(* Logix 5000 project; controller AMANA_DC_PLANT_01 vendor 1 type 14 code 164 rev 31.12; software revision 31.02; part 6 of 9 *)
(* tags used below, declared in another part *)
   badModel : STRING_40;
   Break_1stStation : BOOL;
   firstCharacter : STRING_40;
   Local_Timer : TIMER[10];
   OneShot : DINT;
   ONS_20 : DINT;
   previousSerialNumber : STRING;
   readIndex : DINT;
   tempIndex : DINT;
   writeIndex : DINT;
   DC1_OPCFault : BOOL;
   DC1_to_LN00_Messages : DINT[20];
   DC1_to_LN00_Time_sync_Out : MESSAGE;
   LN00_COUNTS_FROM_IGN_DB_msg : MESSAGE;
   LN00_MainLine_MSG_Out : MESSAGE;
   LN00_Schedule : UDT_Current_Status;
   LN00_SNModel_Array : UDT_SN_Model[50];
   LN00_SNModel_CurrentRead : UDT_SN_Model;
   LN00_SNModel_STR : STRING[10];
   LN00_to_DC1_Main_Messages_6 : DINT[120];
   LN00DFM04 : DINT;
   LN00DFM05 : DINT;
   LN00DFM06 : DINT;
   LN00DFM07 : DINT;
   LN00DFM08 : DINT;
   LN00DFM09 : DINT;
   LN00DFM10 : DINT;
   LN00DFM11 : DINT;
   LN00DFM12 : DINT;
   LN00DFM13 : DINT;
   LN00DFM14 : DINT;
   LN00DFM15 : DINT;
   LN00DFM16 : DINT;
   LN00DFM17 : DINT;
   LN00DFM18 : DINT;
   LN00DFM19 : DINT;
   LN00DFM20 : DINT;
   LN00DFM21 : DINT;
   LN00DFM22 : DINT;
   LN00DFM23 : DINT;
   LN00DFM24 : DINT;
   LN00DFM25 : DINT;
   LN00DFM26 : DINT;
   LN00DFM27 : DINT;
   LN00DFM28 : DINT;
   LN00DFM29 : DINT;
   LN00DFM30 : DINT;
   LN00DFM31 : DINT;
   LN00DFM32 : DINT;
   LN00DFM33 : DINT;
   LN00DFM34 : DINT;
   LN00DFM35 : DINT;
   msg192_reset_timer : TIMER;
   null : STRING;
   OH_Barcode_Model_CLEARPACK : STRING;
   OH_Barcode_Model_DOCKSORTING : STRING;
   OH_Barcode_Model_LN4 : STRING;
   OH_Barcode_Model_LN467MERGE : STRING;
   OH_Barcode_Model_LN6 : STRING;
   OH_Barcode_Model_LN67MERGE : STRING;
   OH_Barcode_Model_LN7 : STRING;
   OH_Barcode_Model_LONGTERMEAST : STRING;
   OH_Barcode_Model_LONGTERMWEST : STRING;
   OH_Barcode_Model_WAREHOUSENORTH : STRING;
   OH_Barcode_Model_WAREHOUSESOUTH : STRING;
   OH_Barcode_Serial_CLEARPACK : STRING;
   OH_Barcode_Serial_DOCKSORTING : STRING;
   OH_Barcode_Serial_LN4 : STRING;
   OH_Barcode_Serial_LN467MERGE : STRING;
   OH_Barcode_Serial_LN6 : STRING;
   OH_Barcode_Serial_LN67MERGE : STRING;
   OH_Barcode_Serial_LN7 : STRING;
   OH_Barcode_Serial_LONGTERMEAST : STRING;
   OH_Barcode_Serial_LONGTERMWEST : STRING;
   OH_Barcode_Serial_WAREHOUSENORTH : STRING;
   OH_Barcode_Serial_WAREHOUSESOUTH : STRING;
   Shift_reset_timer : TIMER;
(* LN00, continued *)

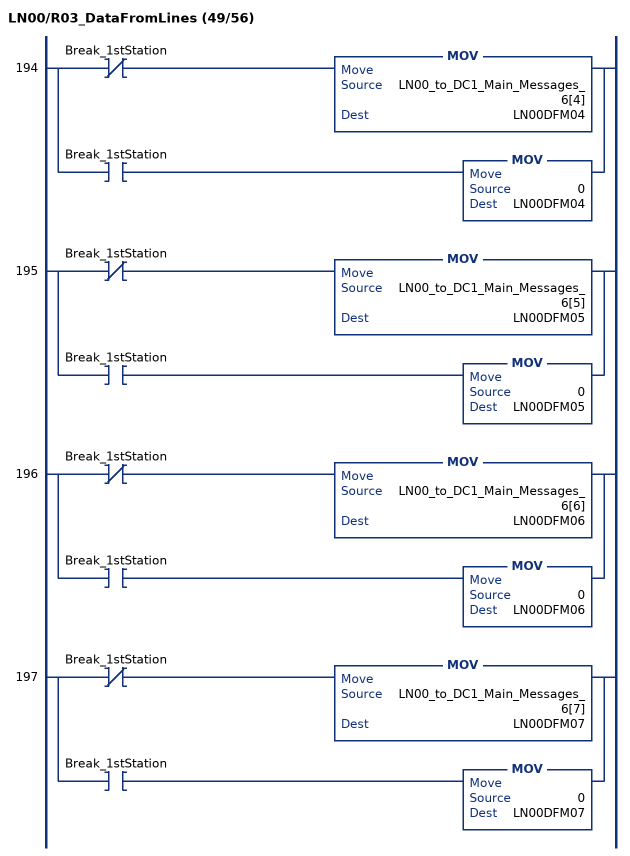
   [picture p95: LN00/R03_DataFromLines rungs 194-197]
   194: [XIO(Break_1stStation) MOV(LN00_to_DC1_Main_Messages_6[4],LN00DFM04) ,XIC(Break_1stStation) MOV(0,LN00DFM04) ];
   195: [XIO(Break_1stStation) MOV(LN00_to_DC1_Main_Messages_6[5],LN00DFM05) ,XIC(Break_1stStation) MOV(0,LN00DFM05) ];
   196: [XIO(Break_1stStation) MOV(LN00_to_DC1_Main_Messages_6[6],LN00DFM06) ,XIC(Break_1stStation) MOV(0,LN00DFM06) ];
   197: [XIO(Break_1stStation) MOV(LN00_to_DC1_Main_Messages_6[7],LN00DFM07) ,XIC(Break_1stStation) MOV(0,LN00DFM07) ];
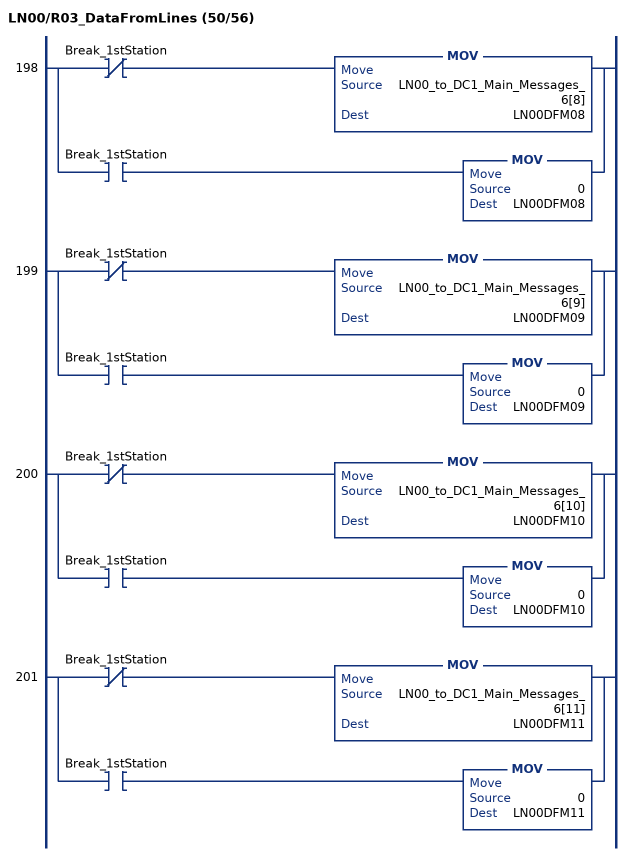
   198: [XIO(Break_1stStation) MOV(LN00_to_DC1_Main_Messages_6[8],LN00DFM08) ,XIC(Break_1stStation) MOV(0,LN00DFM08) ];
   199: [XIO(Break_1stStation) MOV(LN00_to_DC1_Main_Messages_6[9],LN00DFM09) ,XIC(Break_1stStation) MOV(0,LN00DFM09) ];
   200: [XIO(Break_1stStation) MOV(LN00_to_DC1_Main_Messages_6[10],LN00DFM10) ,XIC(Break_1stStation) MOV(0,LN00DFM10) ];
   201: [XIO(Break_1stStation) MOV(LN00_to_DC1_Main_Messages_6[11],LN00DFM11) ,XIC(Break_1stStation) MOV(0,LN00DFM11) ];
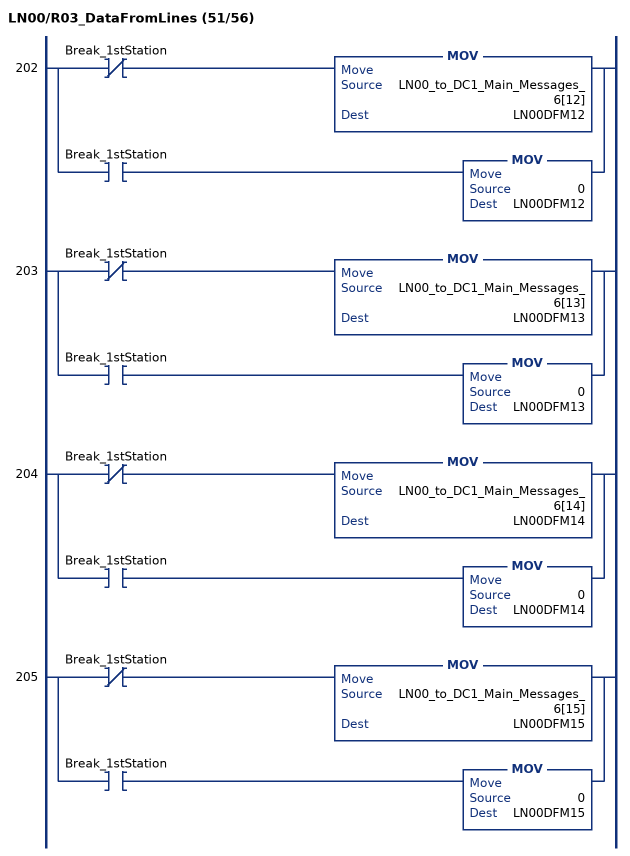
   202: [XIO(Break_1stStation) MOV(LN00_to_DC1_Main_Messages_6[12],LN00DFM12) ,XIC(Break_1stStation) MOV(0,LN00DFM12) ];
   203: [XIO(Break_1stStation) MOV(LN00_to_DC1_Main_Messages_6[13],LN00DFM13) ,XIC(Break_1stStation) MOV(0,LN00DFM13) ];
   204: [XIO(Break_1stStation) MOV(LN00_to_DC1_Main_Messages_6[14],LN00DFM14) ,XIC(Break_1stStation) MOV(0,LN00DFM14) ];
   205: [XIO(Break_1stStation) MOV(LN00_to_DC1_Main_Messages_6[15],LN00DFM15) ,XIC(Break_1stStation) MOV(0,LN00DFM15) ];
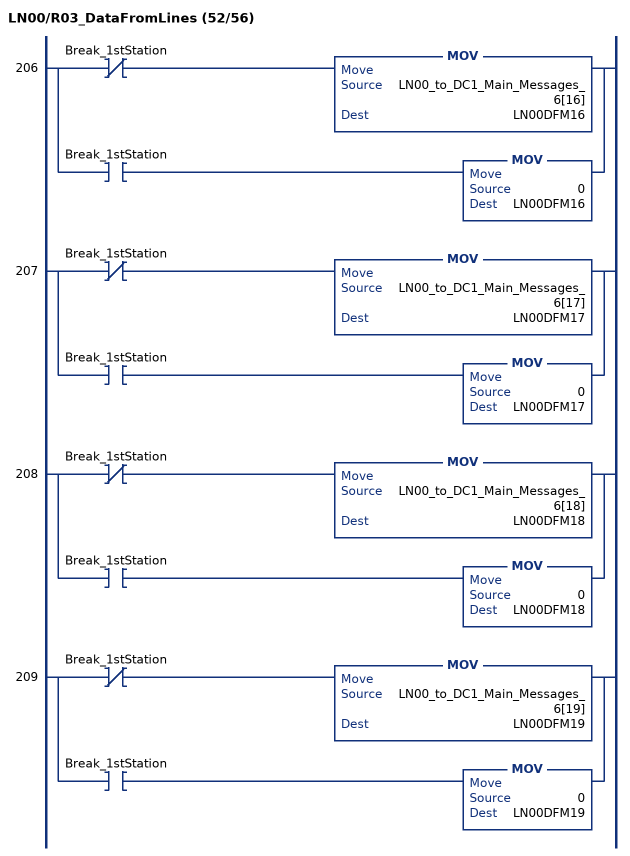
   206: [XIO(Break_1stStation) MOV(LN00_to_DC1_Main_Messages_6[16],LN00DFM16) ,XIC(Break_1stStation) MOV(0,LN00DFM16) ];
   207: [XIO(Break_1stStation) MOV(LN00_to_DC1_Main_Messages_6[17],LN00DFM17) ,XIC(Break_1stStation) MOV(0,LN00DFM17) ];
   208: [XIO(Break_1stStation) MOV(LN00_to_DC1_Main_Messages_6[18],LN00DFM18) ,XIC(Break_1stStation) MOV(0,LN00DFM18) ];
   209: [XIO(Break_1stStation) MOV(LN00_to_DC1_Main_Messages_6[19],LN00DFM19) ,XIC(Break_1stStation) MOV(0,LN00DFM19) ];
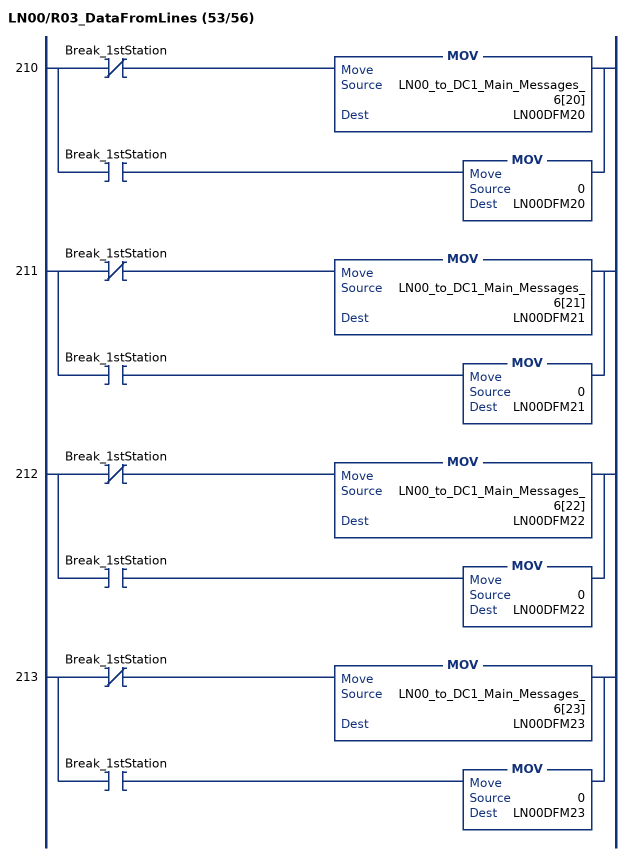
   210: [XIO(Break_1stStation) MOV(LN00_to_DC1_Main_Messages_6[20],LN00DFM20) ,XIC(Break_1stStation) MOV(0,LN00DFM20) ];
   211: [XIO(Break_1stStation) MOV(LN00_to_DC1_Main_Messages_6[21],LN00DFM21) ,XIC(Break_1stStation) MOV(0,LN00DFM21) ];
   212: [XIO(Break_1stStation) MOV(LN00_to_DC1_Main_Messages_6[22],LN00DFM22) ,XIC(Break_1stStation) MOV(0,LN00DFM22) ];
   213: [XIO(Break_1stStation) MOV(LN00_to_DC1_Main_Messages_6[23],LN00DFM23) ,XIC(Break_1stStation) MOV(0,LN00DFM23) ];
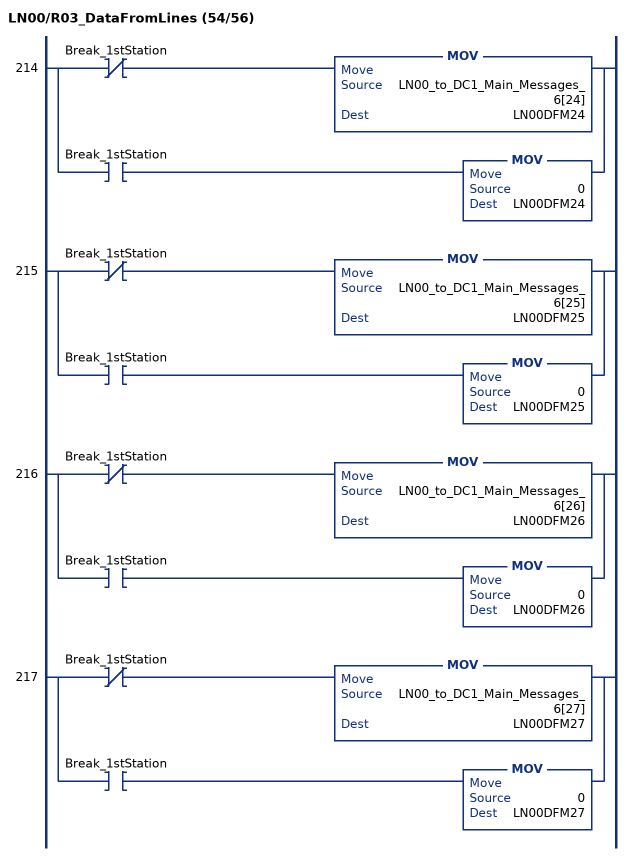
   214: [XIO(Break_1stStation) MOV(LN00_to_DC1_Main_Messages_6[24],LN00DFM24) ,XIC(Break_1stStation) MOV(0,LN00DFM24) ];
   215: [XIO(Break_1stStation) MOV(LN00_to_DC1_Main_Messages_6[25],LN00DFM25) ,XIC(Break_1stStation) MOV(0,LN00DFM25) ];
   216: [XIO(Break_1stStation) MOV(LN00_to_DC1_Main_Messages_6[26],LN00DFM26) ,XIC(Break_1stStation) MOV(0,LN00DFM26) ];
   217: [XIO(Break_1stStation) MOV(LN00_to_DC1_Main_Messages_6[27],LN00DFM27) ,XIC(Break_1stStation) MOV(0,LN00DFM27) ];
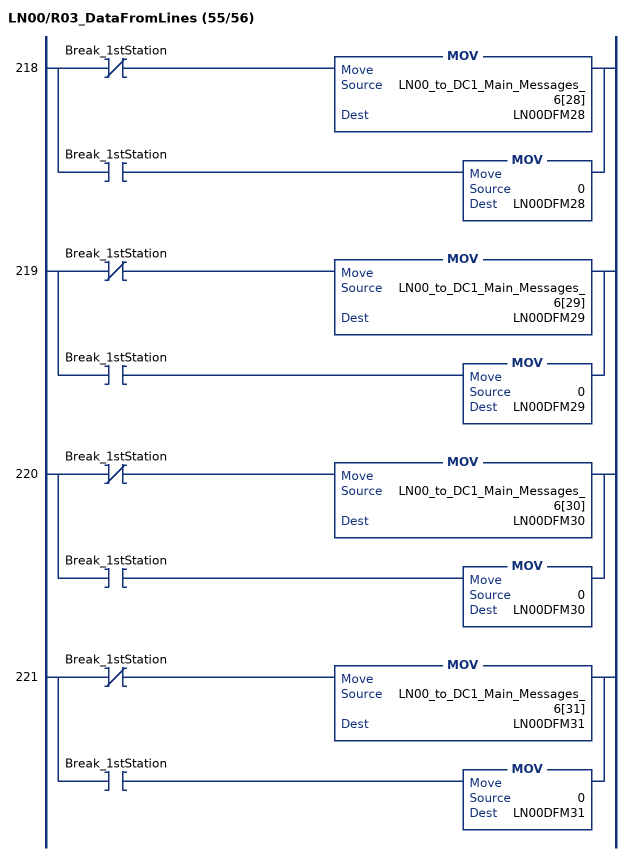
   218: [XIO(Break_1stStation) MOV(LN00_to_DC1_Main_Messages_6[28],LN00DFM28) ,XIC(Break_1stStation) MOV(0,LN00DFM28) ];
   219: [XIO(Break_1stStation) MOV(LN00_to_DC1_Main_Messages_6[29],LN00DFM29) ,XIC(Break_1stStation) MOV(0,LN00DFM29) ];
   220: [XIO(Break_1stStation) MOV(LN00_to_DC1_Main_Messages_6[30],LN00DFM30) ,XIC(Break_1stStation) MOV(0,LN00DFM30) ];
   221: [XIO(Break_1stStation) MOV(LN00_to_DC1_Main_Messages_6[31],LN00DFM31) ,XIC(Break_1stStation) MOV(0,LN00DFM31) ];
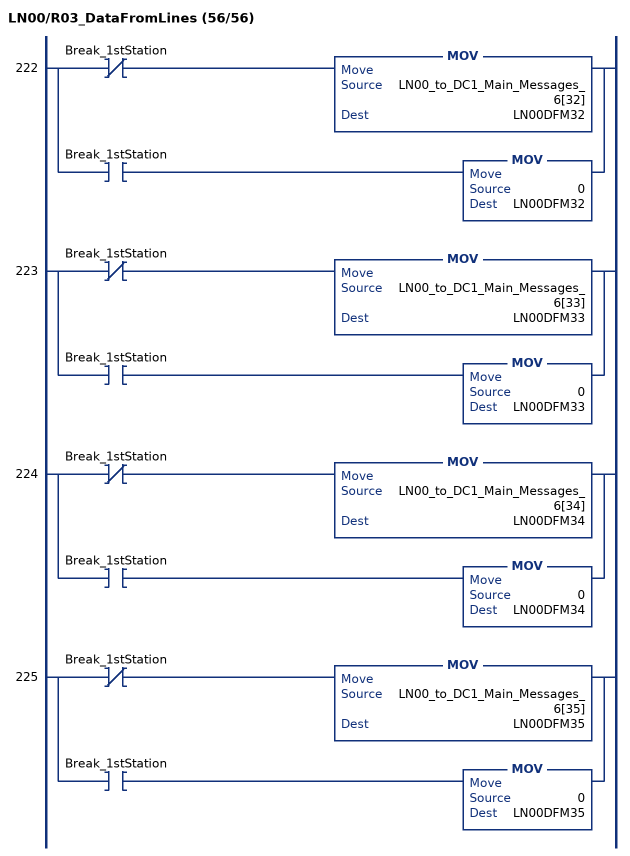
   222: [XIO(Break_1stStation) MOV(LN00_to_DC1_Main_Messages_6[32],LN00DFM32) ,XIC(Break_1stStation) MOV(0,LN00DFM32) ];
   223: [XIO(Break_1stStation) MOV(LN00_to_DC1_Main_Messages_6[33],LN00DFM33) ,XIC(Break_1stStation) MOV(0,LN00DFM33) ];
   224: [XIO(Break_1stStation) MOV(LN00_to_DC1_Main_Messages_6[34],LN00DFM34) ,XIC(Break_1stStation) MOV(0,LN00DFM34) ];
   225: [XIO(Break_1stStation) MOV(LN00_to_DC1_Main_Messages_6[35],LN00DFM35) ,XIC(Break_1stStation) MOV(0,LN00DFM35) ];
END_ROUTINE

ROUTINE R04_DataToLines   (* ladder *)
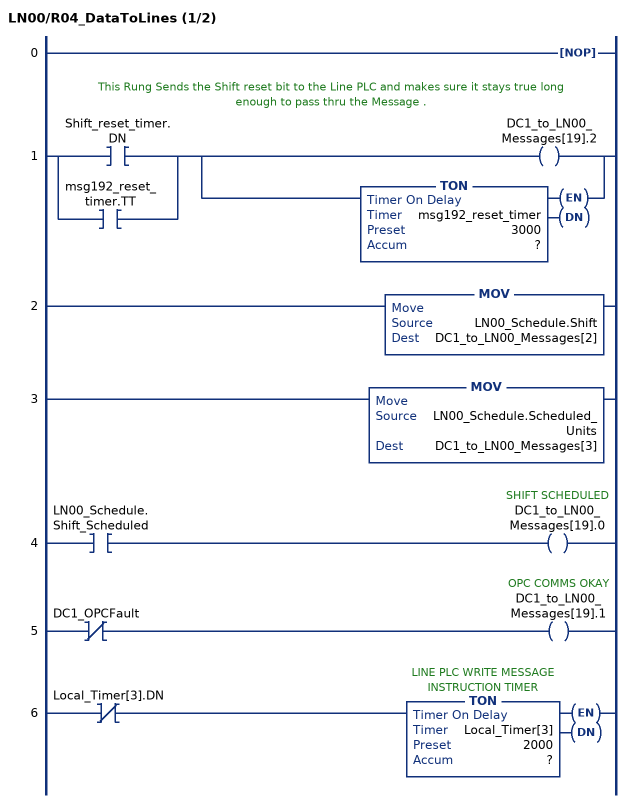
   0: NOP();
   // This Rung Sends the Shift reset bit to the Line PLC and makes sure it stays true long enough to pass thru the Message .
   1: [XIC(Shift_reset_timer.DN) ,XIC(msg192_reset_timer.TT) ][OTE(DC1_to_LN00_Messages[19].2) ,TON(msg192_reset_timer,?,?) ];
   2: MOV(LN00_Schedule.Shift,DC1_to_LN00_Messages[2]);
   3: MOV(LN00_Schedule.Scheduled_Units,DC1_to_LN00_Messages[3]);
   4: XIC(LN00_Schedule.Shift_Scheduled)OTE(DC1_to_LN00_Messages[19].0);
   5: XIO(DC1_OPCFault)OTE(DC1_to_LN00_Messages[19].1);
   6: XIO(Local_Timer[3].DN)TON(Local_Timer[3],?,?);
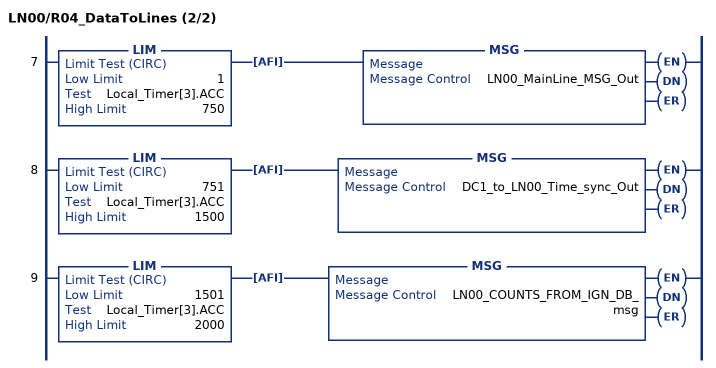
   7: LIM(1,Local_Timer[3].ACC,750)AFI()MSG(LN00_MainLine_MSG_Out);
   8: LIM(751,Local_Timer[3].ACC,1500)AFI()MSG(DC1_to_LN00_Time_sync_Out);
   9: LIM(1501,Local_Timer[3].ACC,2000)AFI()MSG(LN00_COUNTS_FROM_IGN_DB_msg);
END_ROUTINE

ROUTINE R05_SNModel_Manager   (* ladder *)
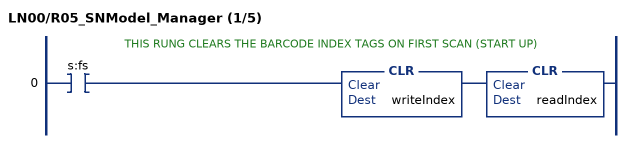
   // THIS RUNG CLEARS THE BARCODE INDEX TAGS ON FIRST SCAN (START UP)
   0: XIC(s:fs)CLR(writeIndex)CLR(readIndex);
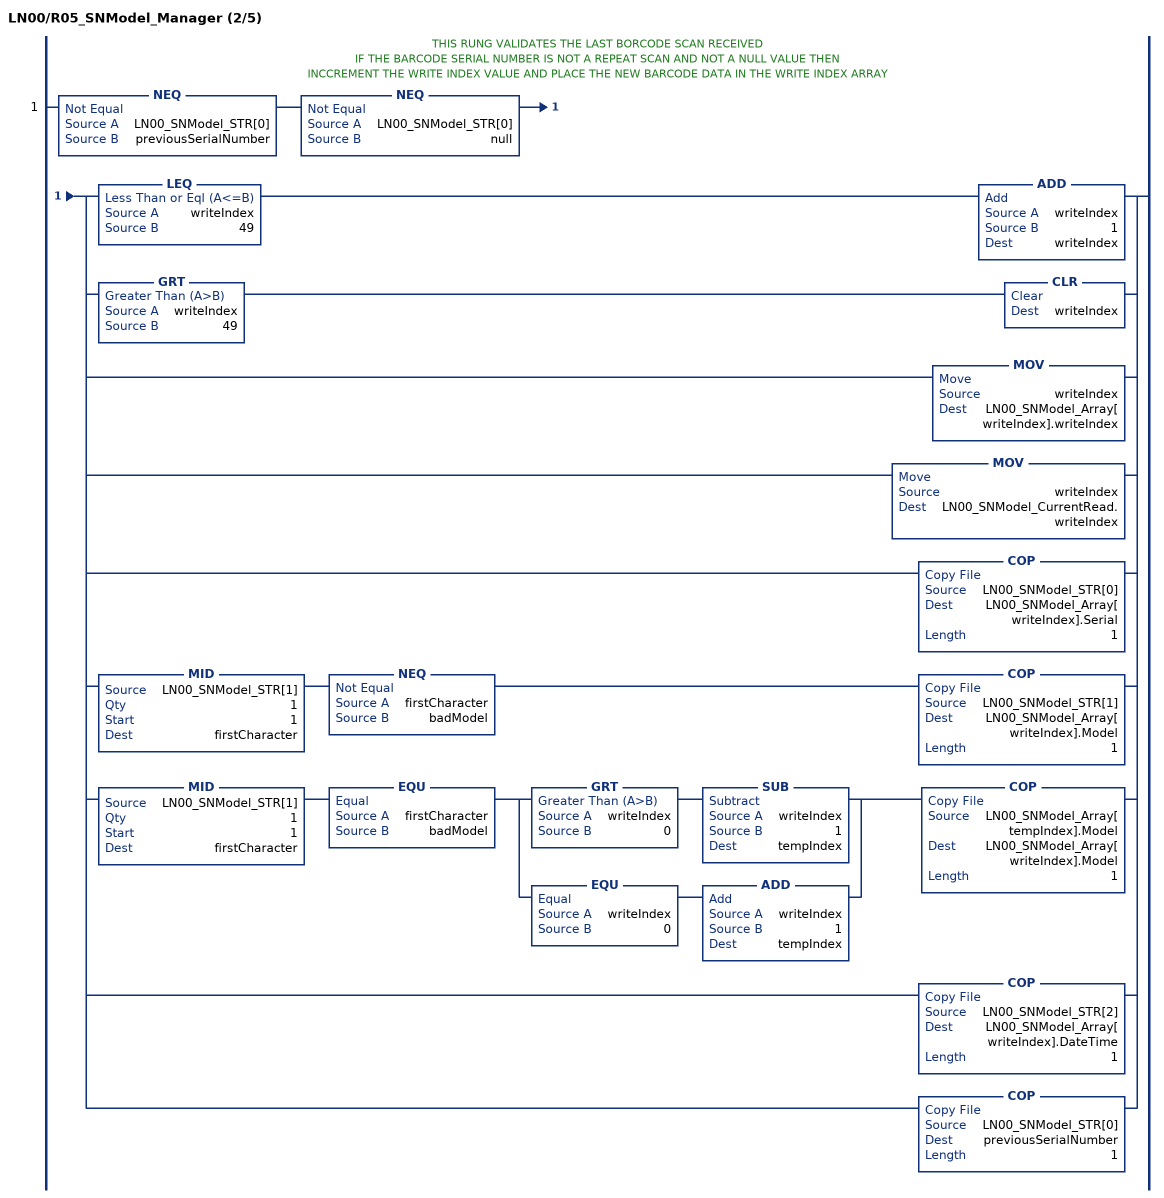
   // THIS RUNG VALIDATES THE LAST BORCODE SCAN RECEIVED
   // IF THE BARCODE SERIAL NUMBER IS NOT A REPEAT SCAN AND NOT A NULL VALUE THEN
   // INCCREMENT THE WRITE INDEX VALUE AND PLACE THE NEW BARCODE DATA IN THE WRITE INDEX ARRAY
   1: NEQ(LN00_SNModel_STR[0],previousSerialNumber)NEQ(LN00_SNModel_STR[0],null)[[LEQ(writeIndex,49) ADD(writeIndex,1,writeIndex) ,GRT(writeIndex,49) CLR(writeIndex) ,MOV(writeIndex,LN00_SNModel_Array[writeIndex].writeIndex) ,MOV(writeIndex,LN00_SNModel_CurrentRead.writeIndex) ,COP(LN00_SNModel_STR[0],LN00_SNModel_Array[writeIndex].Serial,1) ,MID(LN00_SNModel_STR[1],1,1,firstCharacter) NEQ(firstCharacter,badModel) COP(LN00_SNModel_STR[1],LN00_SNModel_Array[writeIndex].Model,1) ,MID(LN00_SNModel_STR[1],1,1,firstCharacter) EQU(firstCharacter,badModel) [GRT(writeIndex,0) SUB(writeIndex,1,tempIndex) ,EQU(writeIndex,0) ADD(writeIndex,1,tempIndex) ] COP(LN00_SNModel_Array[tempIndex].Model,LN00_SNModel_Array[writeIndex].Model,1) ,COP(LN00_SNModel_STR[2],LN00_SNModel_Array[writeIndex].DateTime,1) ] ,COP(LN00_SNModel_STR[0],previousSerialNumber,1) ];
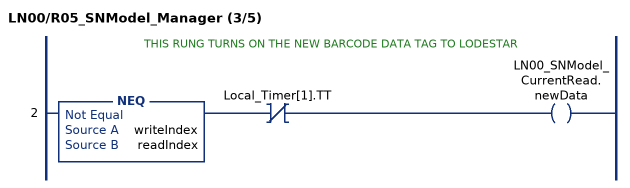
   // THIS RUNG TURNS ON THE NEW BARCODE DATA TAG TO LODESTAR
   2: NEQ(writeIndex,readIndex)XIO(Local_Timer[1].TT)OTE(LN00_SNModel_CurrentRead.newData);
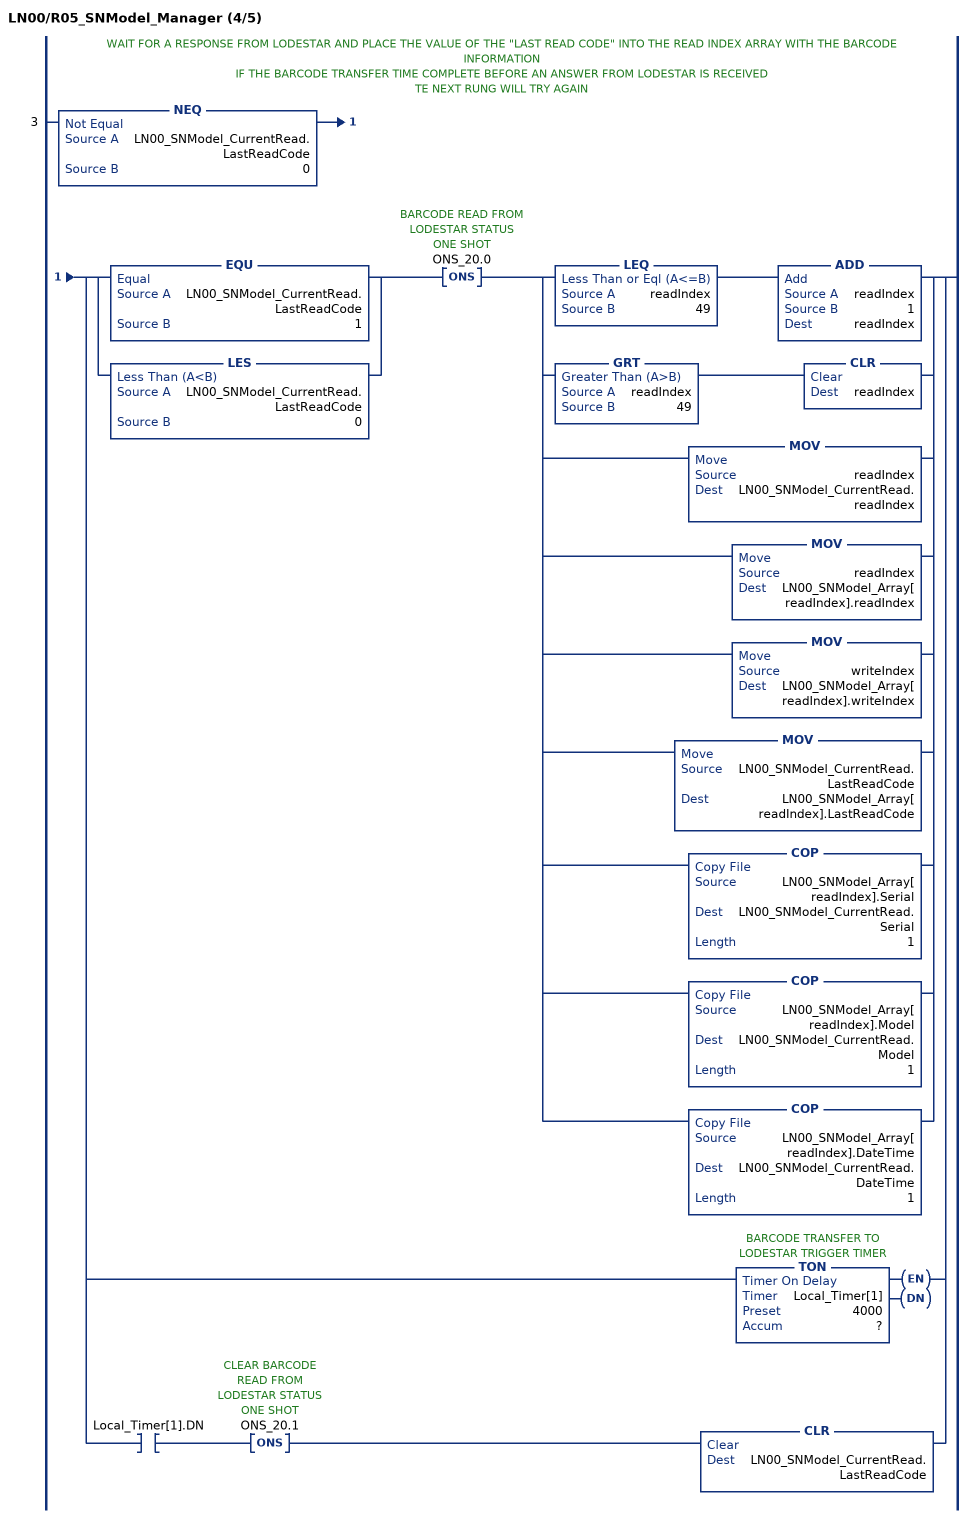
   // WAIT FOR A RESPONSE FROM LODESTAR AND PLACE THE VALUE OF THE "LAST READ CODE" INTO THE READ INDEX ARRAY WITH THE BARCODE INFORMATION
   // IF THE BARCODE TRANSFER TIME COMPLETE BEFORE AN ANSWER FROM LODESTAR IS RECEIVED
   // TE NEXT RUNG WILL TRY AGAIN
   3: NEQ(LN00_SNModel_CurrentRead.LastReadCode,0)[[EQU(LN00_SNModel_CurrentRead.LastReadCode,1) ,LES(LN00_SNModel_CurrentRead.LastReadCode,0) ] ONS(ONS_20.0) [LEQ(readIndex,49) ADD(readIndex,1,readIndex) ,GRT(readIndex,49) CLR(readIndex) ,MOV(readIndex,LN00_SNModel_CurrentRead.readIndex) ,MOV(readIndex,LN00_SNModel_Array[readIndex].readIndex) ,MOV(writeIndex,LN00_SNModel_Array[readIndex].writeIndex) ,MOV(LN00_SNModel_CurrentRead.LastReadCode,LN00_SNModel_Array[readIndex].LastReadCode) ,COP(LN00_SNModel_Array[readIndex].Serial,LN00_SNModel_CurrentRead.Serial,1) ,COP(LN00_SNModel_Array[readIndex].Model,LN00_SNModel_CurrentRead.Model,1) ,COP(LN00_SNModel_Array[readIndex].DateTime,LN00_SNModel_CurrentRead.DateTime,1) ] ,[TON(Local_Timer[1],?,?) ,XIC(Local_Timer[1].DN) ONS(ONS_20.1) CLR(LN00_SNModel_CurrentRead.LastReadCode) ] ];
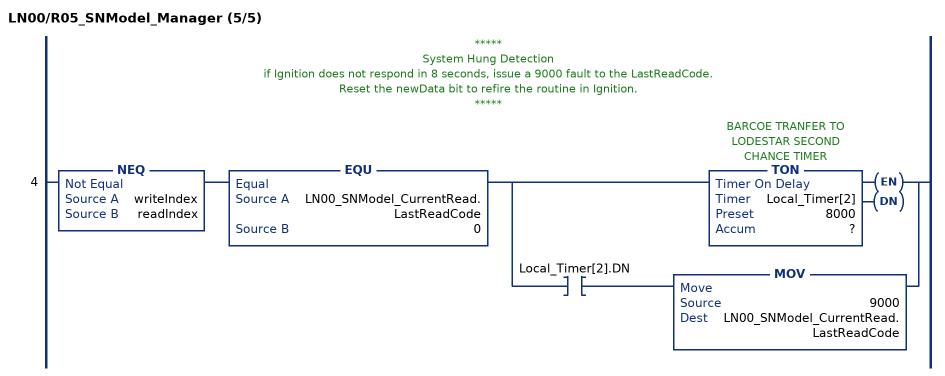
   // *****
   // System Hung Detection
   // if Ignition does not respond in 8 seconds, issue a 9000 fault to the LastReadCode.
   // Reset the newData bit to refire the routine in Ignition.
   // *****
   4: NEQ(writeIndex,readIndex)EQU(LN00_SNModel_CurrentRead.LastReadCode,0)[TON(Local_Timer[2],?,?) ,XIC(Local_Timer[2].DN) MOV(9000,LN00_SNModel_CurrentRead.LastReadCode) ];
END_ROUTINE
END_PROGRAM

PROGRAM OH_BARCODE_SCAN   (* main routine R00_Main *)
VAR
   Barcode_Longest : DINT := 24;
   Barcode_Shortest : DINT := 20;
   Comma : STRING := ',';
   Counters : COUNTER[16] := ([1].PRE := 3, [2].DN := 1, [3].DN := 1, [4].DN := 1, [5].DN := 1, [6].DN := 1);
        [1]   // ClearPack MSG 1 Error Counter
   MSG_Enable : DINT := 34;
   MSG_ONS : DINT := 4;
   MSG_Steps : DINT := 2;
   NULL_String : STRING;
   PRE_SET_COMMA_POSITION_1 : DINT := 12;
   SCANNER_ClearPack_DATA : Keyence_2_Barcode := (Trigger_Timer.PRE := 500, Barcode_ReadIsSuccess := 1, Barcode_Raw := 'WRB322DMBM 03,KC1814086', Barcode_Comma_Position := 14, Barcode_1_Length := 13, Barcode_2_Length := 9, Barcode_2_Start := 15, Barcode_1_String := 'WRB322DMBM 03', Barcode_2_String := 'KC1814086', Barcode_SRReaderReady := 1);
   SCANNER_DOCKSORTING_DATA : Keyence_2_Barcode := (Trigger_Timer.PRE := 200, Trigger_Timer.EN := 1, Trigger_Timer.DN := 1, Barcode_SRTrigger := 1, Barcode_Comma_Position := 10, Barcode_1_Length := 9, Barcode_2_Length := 13, Barcode_2_Start := 11, PlaceHolder_ConveyorRunning := 1, OneShot := 1);
   SCANNER_LN467MERGE_DATA : Keyence_2_Barcode := (Trigger_Timer.PRE := 200, Trigger_Timer.ACC := 200, OneShot := 1);
   SCANNER_LN4_DATA : Keyence_2_Barcode := (Trigger_Timer.PRE := 200, Trigger_Timer.ACC := 200, OneShot := 1);
   SCANNER_LN67MERGE_DATA : Keyence_2_Barcode := (Trigger_Timer.PRE := 200, Trigger_Timer.ACC := 200, OneShot := 1);
   SCANNER_LN6_DATA : Keyence_2_Barcode := (Trigger_Timer.PRE := 200, Trigger_Timer.ACC := 200, OneShot := 1);
   SCANNER_LN7_DATA : Keyence_2_Barcode := (Trigger_Timer.PRE := 200, Trigger_Timer.ACC := 200, OneShot := 1);
   SCANNER_LONGTERMEAST_DATA : Keyence_2_Barcode := (Trigger_Timer.PRE := 200, Trigger_Timer.ACC := 200, OneShot := 1);
   SCANNER_LONGTERMWEST_DATA : Keyence_2_Barcode := (Trigger_Timer.PRE := 200, Trigger_Timer.ACC := 200, OneShot := 1);
   SCANNER_WAREHOUSENORTH_DATA : Keyence_2_Barcode := (Trigger_Timer.PRE := 200, Trigger_Timer.ACC := 200, OneShot := 1);
   SCANNER_WAREHOUSESOUTH_DATA : Keyence_2_Barcode := (Trigger_Timer.PRE := 200, Trigger_Timer.ACC := 200, OneShot := 1);
   Test_Bits : DINT := 2051;
   Timer_MSG_Interval : TIMER := (PRE := 500);
END_VAR

ROUTINE R00_Main   (* ladder *)
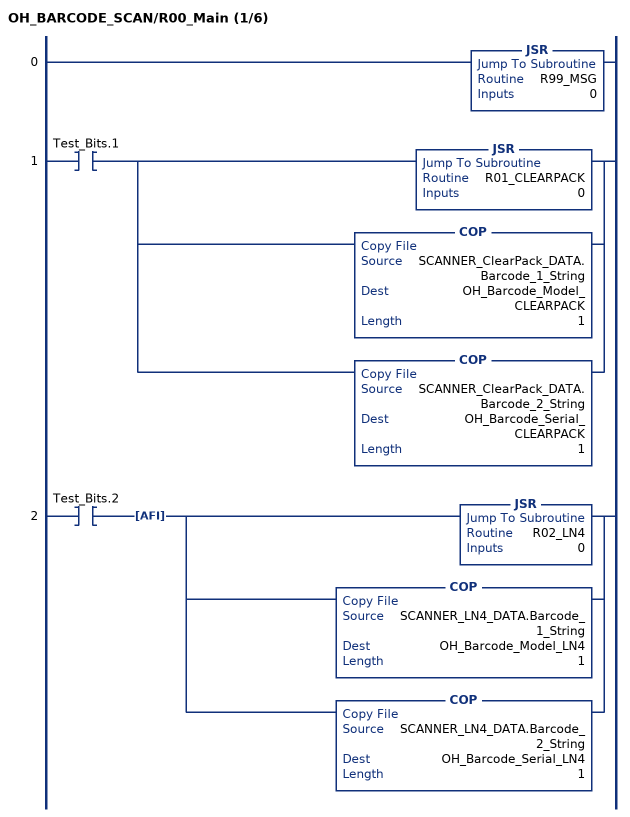
   0: JSR(R99_MSG,0);
   1: XIC(Test_Bits.1)[JSR(R01_CLEARPACK,0) ,COP(SCANNER_ClearPack_DATA.Barcode_1_String,OH_Barcode_Model_CLEARPACK,1) ,COP(SCANNER_ClearPack_DATA.Barcode_2_String,OH_Barcode_Serial_CLEARPACK,1) ];
   2: XIC(Test_Bits.2)AFI()[JSR(R02_LN4,0) ,COP(SCANNER_LN4_DATA.Barcode_1_String,OH_Barcode_Model_LN4,1) ,COP(SCANNER_LN4_DATA.Barcode_2_String,OH_Barcode_Serial_LN4,1) ];
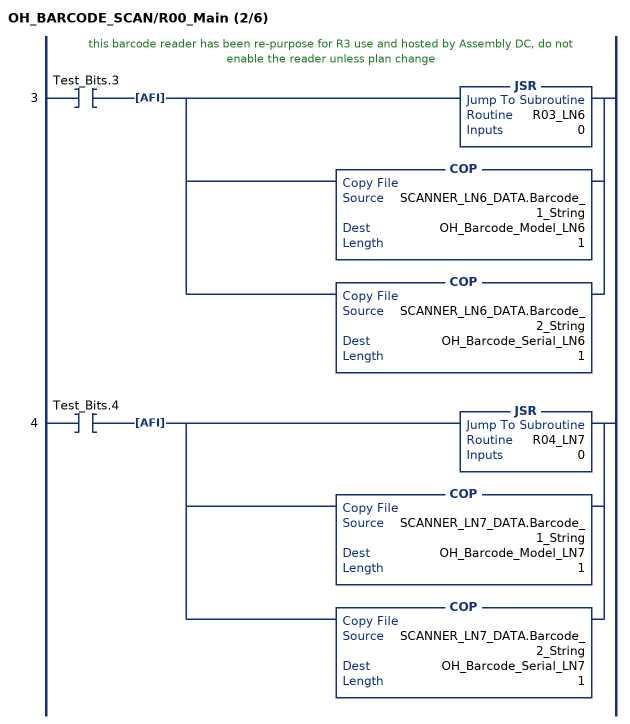
   // this barcode reader has been re-purpose for R3 use and hosted by Assembly DC, do not enable the reader unless plan change
   3: XIC(Test_Bits.3)AFI()[JSR(R03_LN6,0) ,COP(SCANNER_LN6_DATA.Barcode_1_String,OH_Barcode_Model_LN6,1) ,COP(SCANNER_LN6_DATA.Barcode_2_String,OH_Barcode_Serial_LN6,1) ];
   4: XIC(Test_Bits.4)AFI()[JSR(R04_LN7,0) ,COP(SCANNER_LN7_DATA.Barcode_1_String,OH_Barcode_Model_LN7,1) ,COP(SCANNER_LN7_DATA.Barcode_2_String,OH_Barcode_Serial_LN7,1) ];
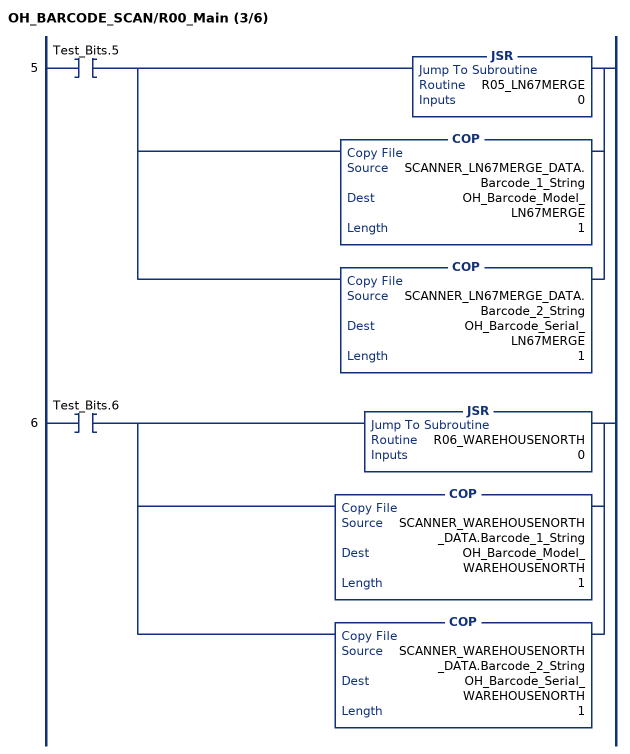
   5: XIC(Test_Bits.5)[JSR(R05_LN67MERGE,0) ,COP(SCANNER_LN67MERGE_DATA.Barcode_1_String,OH_Barcode_Model_LN67MERGE,1) ,COP(SCANNER_LN67MERGE_DATA.Barcode_2_String,OH_Barcode_Serial_LN67MERGE,1) ];
   6: XIC(Test_Bits.6)[JSR(R06_WAREHOUSENORTH,0) ,COP(SCANNER_WAREHOUSENORTH_DATA.Barcode_1_String,OH_Barcode_Model_WAREHOUSENORTH,1) ,COP(SCANNER_WAREHOUSENORTH_DATA.Barcode_2_String,OH_Barcode_Serial_WAREHOUSENORTH,1) ];
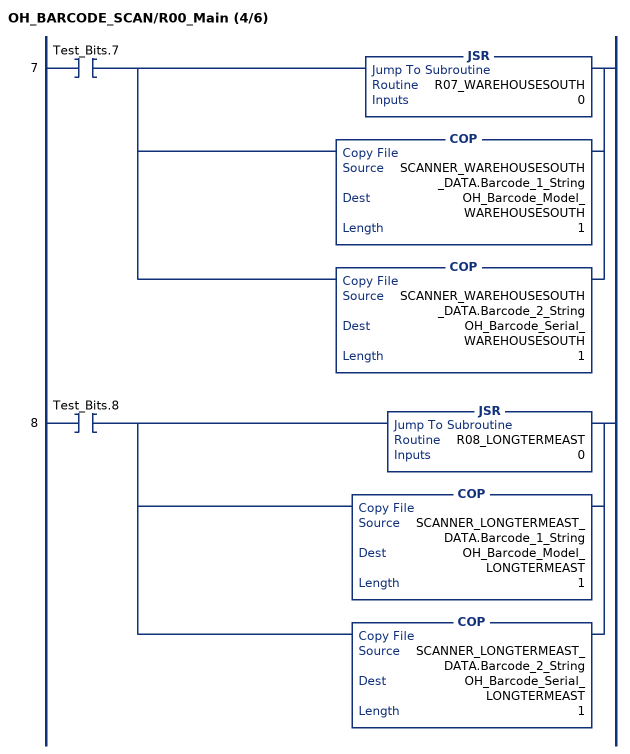
   7: XIC(Test_Bits.7)[JSR(R07_WAREHOUSESOUTH,0) ,COP(SCANNER_WAREHOUSESOUTH_DATA.Barcode_1_String,OH_Barcode_Model_WAREHOUSESOUTH,1) ,COP(SCANNER_WAREHOUSESOUTH_DATA.Barcode_2_String,OH_Barcode_Serial_WAREHOUSESOUTH,1) ];
   8: XIC(Test_Bits.8)[JSR(R08_LONGTERMEAST,0) ,COP(SCANNER_LONGTERMEAST_DATA.Barcode_1_String,OH_Barcode_Model_LONGTERMEAST,1) ,COP(SCANNER_LONGTERMEAST_DATA.Barcode_2_String,OH_Barcode_Serial_LONGTERMEAST,1) ];
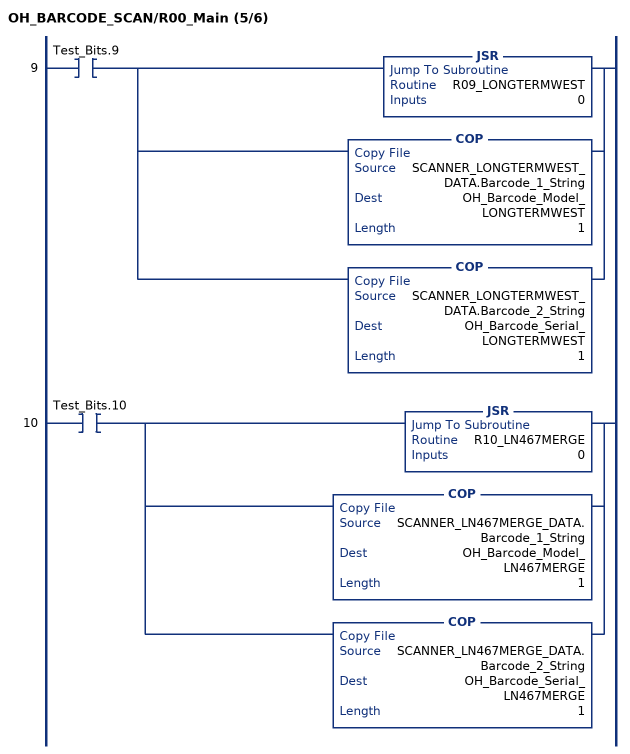
   9: XIC(Test_Bits.9)[JSR(R09_LONGTERMWEST,0) ,COP(SCANNER_LONGTERMWEST_DATA.Barcode_1_String,OH_Barcode_Model_LONGTERMWEST,1) ,COP(SCANNER_LONGTERMWEST_DATA.Barcode_2_String,OH_Barcode_Serial_LONGTERMWEST,1) ];
   10: XIC(Test_Bits.10)[JSR(R10_LN467MERGE,0) ,COP(SCANNER_LN467MERGE_DATA.Barcode_1_String,OH_Barcode_Model_LN467MERGE,1) ,COP(SCANNER_LN467MERGE_DATA.Barcode_2_String,OH_Barcode_Serial_LN467MERGE,1) ];
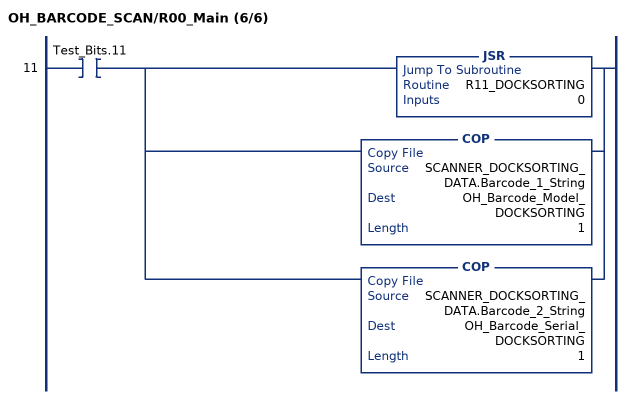
   11: XIC(Test_Bits.11)[JSR(R11_DOCKSORTING,0) ,COP(SCANNER_DOCKSORTING_DATA.Barcode_1_String,OH_Barcode_Model_DOCKSORTING,1) ,COP(SCANNER_DOCKSORTING_DATA.Barcode_2_String,OH_Barcode_Serial_DOCKSORTING,1) ];
END_ROUTINE
